{attribute addProperty BoxType "EJ3318-0000-0017"}
{attribute addProperty Id "TC_ChannelAT %I*ARRAY[0..7] OF TC_Channel_17AE08DB256320RTD_Inputs_ChannelAT %I*ARRAY[0..1] OF RTD_Inputs_Channel_17AE08DB6480WcStateAT %I*WcState_F855686C1620InfoDataAT %I*InfoData_BC63D37F80100"}
{attribute addProperty CRC "3609340602"}
{attribute addProperty SizeInBites "416"}
{attribute addProperty SizeInBytes "52"}
TYPE EJ3318_513179EA :
STRUCT
	{attribute addProperty Name "TC_Channel"}
	TC_Channel : ARRAY[0..7] OF TC_Channel_17AE08DB;
	{attribute addProperty Name "RTD_Inputs_Channel"}
	RTD_Inputs_Channel : ARRAY[0..1] OF RTD_Inputs_Channel_17AE08DB;
	{attribute addProperty Name "WcState"}
	WcState : WcState_F855686C;
	{attribute addProperty Name "InfoData"}
	InfoData : InfoData_BC63D37F;
END_STRUCT
END_TYPE

(* stored: Version 1.2.0.0, ProductVersion 3.1.4024.9
   DUT EJ3318_513179EA: Id {83b24bec-c157-4c72-ad55-0f21d83df7d5} *)
